{attribute 'analysis' := '-33'}
FUNCTION_BLOCK FB_XTES_Flowswitch
VAR_OUTPUT
    {attribute 'pytmc' := '
        pv: FLOW_OK
        field: ZNAM LOW
        field: ONAM OK
    '}
    bFlowOk AT %I*: BOOL;
END_VAR

END_FUNCTION_BLOCK

(* stored: Version 1.1.0.1
   POU FB_XTES_Flowswitch: Id {8cdc81d2-8d66-4efc-bd9f-1d19d105030f}, SpecialFunc None *)
